FUNCTION_BLOCK Delay
VAR_OUTPUT
	Delay_Done	: BOOL;
END_VAR
VAR
	T			: LREAL :=10;
END_VAR

METHOD Delay_02s
VAR_INPUT
	Drive_Delay 		: BOOL;			//延迟程序使能信号
END_VAR
// =======================延迟程序==========================

IF Drive_Delay THEN
	T := T-0.01;
END_IF

IF T<=0 THEN
	Drive_Delay :=0;	
	T :=1;
	Delay_Done :=1;
END_IF
END_METHOD

END_FUNCTION_BLOCK

(* stored: Version 1.1.0.1, ProductVersion 3.1.4020.12
   POU Delay: Id {9b91272d-9848-4c41-8af9-1af6a2bdd545}, SpecialFunc None
   Method Delay_02s: Id {f507e41f-ba7a-41ca-a277-53236a669a3d} *)
